// TwinCAT 3 PLC project LF_System_PLC
// ProgramVersion: 3.1.4026.22
// CompilerDefines: VISU_USEPROPERTYINFO
// libraries:
//   Tc2_MC2, * (Beckhoff Automation GmbH)
//   Tc2_Standard, * (Beckhoff Automation GmbH)
//   Tc2_System, * (Beckhoff Automation GmbH)
//   Tc3_IotBase, * (Beckhoff Automation GmbH)
//   VisuSymbols, 4.5.0.0 (System)
// project tree:
//   / GlobalTextList.TcGTLO (not stored), PlcTask.TcTTO (not stored), Visualization Manager.TcVMO (not stored)
//   GVLs/ GVL_PosKinematic.TcGVL, IFC_HW.TcGVL
//   POUs/Abfüllmodul/ FB_Abfuellmodul.TcPOU, FB_Dispenser.TcPOU (not stored), FB_EZylinder.TcPOU, FB_Vereinzelung.TcPOU (not stored)
//   POUs/ eBetriebszustand.TcDUT, FB_MqttPublisher.TcPOU, FUN_Scale.TcPOU, MAIN.TcPOU
//   POUs/Extruder/ FB_System_FlaschenFullstand.TcPOU, FB_System_Fullstand.TcPOU (not stored)
//   POUs/Förderband/ FB_System_CNV.TcPOU (not stored)
//   POUs/IoT/ FB_MQTT.TcPOU (not stored)
//   POUs/Manipulator/ FB_Manipulator.TcPOU (not stored)
//   POUs/Manipulator/Roboter/ FB_Roboter.TcPOU (not stored), FB_Roboter_Axis.TcPOU, FB_Roboter_E.TcPOU, FB_Roboter_Logik.TcPOU
//   POUs/Statusleuchte/ FB_Ampelleuchte.TcPOU, FB_Blinklicht.TcPOU
//   POUs/Transport/ FB_Foerderband.TcPOU, FB_Transport.TcPOU, FB_Transport_A.TcPOU, FB_Transport_E.TcPOU, FB_Transport_Logik.TcPOU
//   POUs/Vereinzelung/ FB_SpeicherRohr.TcPOU (not stored), FB_System_Vereinzelung.TcPOU (not stored)
//   VISUs/ Visualization.TcVIS
// real-time tasks:
//   TASK PlcTask: cycle T#10ms, priority 21, ADS port 350
//   TASK PlcTask1: cycle T#10ms, priority 22, ADS port 351
// motion (NC):
//   TASK NC-Task 1 SAF: cycle T#2ms, priority 4, ADS port 501
//   TASK NC-Task 1 SVB: cycle T#10ms, priority 8, ADS port 511
//   AXIS Band (id 1)
//     OtherSettings: AllowMotionCmdToSlave=true
//     encoder EncType=1
//     drive DrvType=5
//       Analog: TorqueSetpointScale=10, ScaleFactorActTorque=0.1
//       TimeComp: TaskDelayCycles=1
//     controller CtrType=1
//       CtrPara: PriorControlFactor=1
//         Observer: BandWidth=20
//   AXIS Extruder1 (id 2)
//     OtherSettings: AllowMotionCmdToSlave=true
//     encoder EncType=1
//     drive DrvType=5
//       Analog: TorqueSetpointScale=10, ScaleFactorActTorque=0.1
//       TimeComp: TaskDelayCycles=1
//     controller CtrType=1
//       CtrPara: PriorControlFactor=1
//         Observer: BandWidth=20
//   AXIS Extruder2 (id 3)
//     OtherSettings: AllowMotionCmdToSlave=true
//     encoder EncType=1
//     drive DrvType=5
//       Analog: TorqueSetpointScale=10, ScaleFactorActTorque=0.1
//       TimeComp: TaskDelayCycles=1
//     controller CtrType=1
//       CtrPara: PriorControlFactor=1
//         Observer: BandWidth=20
//   AXIS Extruder3 (id 4)
//     OtherSettings: AllowMotionCmdToSlave=true
//     encoder EncType=1
//     drive DrvType=5
//       Analog: TorqueSetpointScale=10, ScaleFactorActTorque=0.1
//       TimeComp: TaskDelayCycles=1
//     controller CtrType=1
//       CtrPara: PriorControlFactor=1
//         Observer: BandWidth=20
//   AXIS ManX (id 5)
//     OtherSettings: AllowMotionCmdToSlave=true
//     encoder EncType=1
//     drive DrvType=5
//       Analog: TorqueSetpointScale=10, ScaleFactorActTorque=0.1
//       TimeComp: TaskDelayCycles=1
//     controller CtrType=1
//       CtrPara: PriorControlFactor=1
//         Observer: BandWidth=20
//   AXIS ManY (id 6)
//     OtherSettings: AllowMotionCmdToSlave=true
//     encoder EncType=1
//     drive DrvType=5
//       Analog: TorqueSetpointScale=10, ScaleFactorActTorque=0.1
//       TimeComp: TaskDelayCycles=1
//     controller CtrType=1
//       CtrPara: PriorControlFactor=1
//         Observer: BandWidth=20
//   AXIS ManZ (id 7)
//     OtherSettings: AllowMotionCmdToSlave=true
//     encoder EncType=1
//     drive DrvType=5
//       Analog: TorqueSetpointScale=10, ScaleFactorActTorque=0.1
//       TimeComp: TaskDelayCycles=1
//     controller CtrType=1
//       CtrPara: PriorControlFactor=1
//         Observer: BandWidth=20
//   AXIS ManG (id 8)
//     OtherSettings: AllowMotionCmdToSlave=true
//     encoder EncType=1
//     drive DrvType=5
//       Analog: TorqueSetpointScale=10, ScaleFactorActTorque=0.1
//       TimeComp: TaskDelayCycles=1
//     controller CtrType=1
//       CtrPara: PriorControlFactor=1
//         Observer: BandWidth=20
// variable links:
//   LF_System_PLC/LF_System_PLC Instance <-> NC-Task 1 SAF/Axes/Band
//     PlcTask Inputs/IFC_HW.ax_BandMotor.NcToPlc <-> Outputs/ToPlc
//     PlcTask Outputs/IFC_HW.ax_BandMotor.PlcToNc <-> Inputs/FromPlc
//   LF_System_PLC/LF_System_PLC Instance <-> NC-Task 1 SAF/Axes/Extruder1
//     PlcTask Inputs/IFC_HW.ax_Extruder1.NcToPlc <-> Outputs/ToPlc
//     PlcTask Outputs/IFC_HW.ax_Extruder1.PlcToNc <-> Inputs/FromPlc
//   LF_System_PLC/LF_System_PLC Instance <-> NC-Task 1 SAF/Axes/Extruder2
//     PlcTask Inputs/IFC_HW.ax_Extruder2.NcToPlc <-> Outputs/ToPlc
//     PlcTask Outputs/IFC_HW.ax_Extruder2.PlcToNc <-> Inputs/FromPlc
//   LF_System_PLC/LF_System_PLC Instance <-> NC-Task 1 SAF/Axes/Extruder3
//     PlcTask Inputs/IFC_HW.ax_Extruder3.NcToPlc <-> Outputs/ToPlc
//     PlcTask Outputs/IFC_HW.ax_Extruder3.PlcToNc <-> Inputs/FromPlc
//   LF_System_PLC/LF_System_PLC Instance <-> NC-Task 1 SAF/Axes/ManG
//     PlcTask Inputs/IFC_HW.ax_ManG.NcToPlc <-> Outputs/ToPlc
//     PlcTask Outputs/IFC_HW.ax_ManG.PlcToNc <-> Inputs/FromPlc
//   LF_System_PLC/LF_System_PLC Instance <-> NC-Task 1 SAF/Axes/ManX
//     PlcTask Inputs/IFC_HW.ax_ManX.NcToPlc <-> Outputs/ToPlc
//     PlcTask Outputs/IFC_HW.ax_ManX.PlcToNc <-> Inputs/FromPlc
//   LF_System_PLC/LF_System_PLC Instance <-> NC-Task 1 SAF/Axes/ManY
//     PlcTask Inputs/IFC_HW.ax_ManY.NcToPlc <-> Outputs/ToPlc
//     PlcTask Outputs/IFC_HW.ax_ManY.PlcToNc <-> Inputs/FromPlc
//   LF_System_PLC/LF_System_PLC Instance <-> NC-Task 1 SAF/Axes/ManZ
//     PlcTask Inputs/IFC_HW.ax_ManZ.NcToPlc <-> Outputs/ToPlc
//     PlcTask Outputs/IFC_HW.ax_ManZ.PlcToNc <-> Inputs/FromPlc

// ---- POUs/eBetriebszustand.TcDUT
{attribute 'qualified_only'}
{attribute 'strict'}
{attribute 'to_string'}
TYPE eBetriebszustand :
(
	Off        := 0,   // nicht betriebsbereit
	Error      := 1,   // Fehlerbehafteter Stop
	Setup      := 2,   // Wartung
	Warning    := 3,   // nicht fehlerbehafteter, nicht geplanter Stop
	Init       := 4,   // Herstellung Betriebsbereitschaft
	Ready      := 5,   // betriebsbereit
	Production := 6,   // Betrieb
	Done       := 7,   // Betrieb abgeschlossen
	Stop       := 8
);
END_TYPE

// ---- GVLs/GVL_PosKinematic.TcGVL
{attribute 'qualified_only'}
VAR_GLOBAL
	// Home position
	pXhome : REAL := 29;
	pYhome : REAL := 145.5;
	pZhome : REAL := 45;
	
	// Conveyor position
	pXconv : REAL := 29;
	pYconv : REAL := 145.5;
	pZconv : REAL := 130;
	
	//Scale position
	pXscale : REAL := 36;
	pYscale : REAL := 7.5;
	pZscale : REAL := 131.5;
	
	// Heating position
	pXheat : REAL := 218.5;
	pYheat : REAL := 7;
	pZheat : REAL := 159;
	
	// Storage position
	pX1stor : REAL := 107;
	pX2stor : REAL := 158.7;
	pX3stor : REAL := 209.3;
	pX4stor : REAL := 260.3;
	pYstor : REAL := 139;
	pZstor : REAL := 120;
	
	// Z offset height
	pZoff : REAL := 45;
END_VAR

// ---- GVLs/IFC_HW.TcGVL
// In dieser GVL werden alle Variablen deklariert die auf die realen Klemmen zugreifen
VAR_GLOBAL
	
	// Allgemeine Variablen fur MAIN und HMI
		bEnable		AT%I*	: BOOL;			// Enable Factory (HMI Production Umgebung)
		bExecute	AT%I*	: BOOL;			// Startsignal	(Start Knopf Konsole)
		bStop				: BOOL;			// Stop Variable (interne Variable um FB's zu stoppen)
		
	// Station Statusampel	
		bAmpelRot 	AT%Q* 	: BOOL;			// Signal-LED Rot
		bAmpelGelb 	AT%Q* 	: BOOL;			// Signal-LED Gelb
		bAmpelGrun 	AT%Q* 	: BOOL;			// Signal-LED Grun
			
	// Station Vereinzelung
		bEinzelSens1 	AT%I*	: BOOL;					// Separation Sensor 1 (Kammer)
		bEinzelSens2 	AT%I*	: BOOL;					// Separation Sensor 2 (Rohr)
		bEinzelSens3 	AT%I*	: BOOL;					// Separation Sensor 3 (Flasche auf Kopf)
		bR1AKT1 		AT%Q* 	: BOOL := FALSE;		// Relais 1 Aktor 1 (Schleuse Oben öffnen)
		bR2AKT1 		AT%Q* 	: BOOL := TRUE; 		// Relais 2 Aktor 1 (Schleuse Oben schließen)
		bR1AKT2 		AT%Q* 	: BOOL := FALSE;		// Relais 1 Aktor 2 (Schleuse Unten öffne)
		bR2AKT2 		AT%Q* 	: BOOL := TRUE;			// Relais 2 Aktor 2	(Schleuse Unten schließen)
	
	// Station Forderband
		bBandSens1 	AT %I*	: BOOL;		// Forderband Sensor 1 (Extruder 1)
		bBandSens2	AT %I*	: BOOL;		// Forderband Sensor 2 (Extruder 2)
		bBandSens3 	AT %I*	: BOOL;		// Forderband Sensor 3 (Extruder 3)
		bBandSens4 	AT %I*	: BOOL;		// Forderband Sensor 4 (Übergabe Roboter)
		bBandHub1 	AT %Q*	: BOOL;		// Forderband Hubmagnet 1 (Schleuse Extruder 1)
		bBandHub2 	AT %Q*	: BOOL;		// Forderband Hubmagnet 1 (Schleuse Extruder 2)
		bBandHub3 	AT %Q*	: BOOL;		// Forderband Hubmagnet 1 (Schleuse Extruder 3)
		
		ax_Extruder1 	: AXIS_REF;		// Forderband NC-Achse Extruder 1
		ax_Extruder2 	: AXIS_REF;		// Forderband NC-Achse Extruder 2
		ax_Extruder3 	: AXIS_REF;		// Forderband NC-Achse Extruder 3
		ax_BandMotor 	: AXIS_REF;		// Forderband NC-Achse Band
		
		iBandFullmenge1		: INT := 1;	// in Gramm (Soll Füllmenge Extruder 1)
		iBandFullmenge2		: INT := 1;	// in Gramm (Soll Füllmenge Extruder 2)
		iBandFullmenge3		: INT := 1;	// in Gramm (Soll Füllmenge Extruder 3)
		
	//Füllstandsüberwachung
		iFillSens1 AT%I*	: UINT;		// Füllstandssensor im Granulatspeicher 1
		iFillSens2 AT%I*	: UINT;		// Füllstandssensor im Granulatspeicher 2
		iFillSens3 AT%I*	: UINT;		// Füllstandssensor im Granulatspeicher 3
		
		rFillLevelPercent1	: REAL;		// Füllstand im Granulatspeicher 1 in %
		rFillLevelGramm1	: REAL;		// Füllstand im Granulatspeicher 1 in g
		rFillLevelPercent2	: REAL;		// Füllstand im Granulatspeicher 2 in %
		rFillLevelGramm2	: REAL;		// Füllstand im Granulatspeicher 2 in g
		rFillLevelPercent3	: REAL;		// Füllstand im Granulatspeicher 3 in %
		rFillLevelGramm3	: REAL;		// Füllstand im Granulatspeicher 3 in g
		
		rMaxFillLevel 		: REAL := 375;	// Kalibrierter Füllstand für 10% * 10
		
	// Station Waage
		sWaageNachricht		: STRING;	// Nachricht von Wagezelle (fur virtuelle Inbetriebnahme notig)
		bWaageNull			: BOOL;		// TARA Waage (Waage auf Null setzen)
		iWaageMesswert		: INT;		// Messwert der Waage
		
	// Station Behalteridentifikation
		bIdSensorTrager		: BOOL;		// Sensor bei Erkennung eines Datentrager
		sIdNachricht		: STRING;	// Nachricht von RFID-System (fur virtuelle Inbetriebnahme notig)
		sSeriennummer		: STRING;	// Seriennummer RFID-Tag
		
	//Temperierstation
		bVentilator1 	AT %Q*	: BOOL;		// Ventilator 1
		bVentilator2 	AT %Q*	: BOOL;		// Ventilator 2
		bVentilator3 	AT %Q*	: BOOL;		// Ventilator 3
		
		iTempSens1 		AT%I*	: UINT;		// Temperatursensor 1
		iTempSens2 		AT%I*	: UINT;		// Temperatursensor 2
		iHeizpatrone 	AT%Q*	: UINT;		// Heizpatronen
		
		iMaxTemp				: UINT := 5500;		// in °C * 100
		
	// Station Manipulator
		bManEndXmin 		AT%I* 	: BOOL := TRUE;		// Manipulator min Endschalter Achse x
		bManEndYmin 		AT%I* 	: BOOL := TRUE;		// Manipulator min Endschalter Achse y
		bManEndZmin 		AT%I* 	: BOOL := TRUE;		// Manipulator min Endschalter Achse z
		bManEndGmin 		AT%I* 	: BOOL := TRUE;		// Manipulator min Endschalter Achse Gripper
		bManEndXmax 		AT%I* 	: BOOL := TRUE;		// Manipulator max Endschalter Achse x
		bManEndYmax 		AT%I* 	: BOOL := TRUE;		// Manipulator max Endschalter Achse y
		bManEndZmax 		AT%I* 	: BOOL := TRUE;		// Manipulator max Endschalter Achse z
		bManEndGmax 		AT%I* 	: BOOL := TRUE;		// Manipulator max Endschalter Achse Gripper
		bManBrakeZ			AT%Q*	: BOOL := FALSE;	// Bremse Achse z
		
		ax_ManX			: AXIS_REF;			// Manipulator NC-Achse x
		ax_ManY			: AXIS_REF;			// Manipulator NC-Achse y
		ax_ManZ			: AXIS_REF;			// Manipulator NC-Achse z
		ax_ManG			: AXIS_REF; 		// Manipulator NC-Achse Gripper
		
		bGripperClosed		AT%Q*	: BOOL; 			// signal if gripper is closed ONLY USED IN SIM
			// --- Für die Unity-Simulation (TeachingFactory) benötigt ---
	BandExtruder1_Enable AT%Q* : BOOL;
	BandExtruder1_Velocity AT%Q* : LREAL;
	BandExtruder2_Enable AT%Q* : BOOL;
	BandExtruder2_Velocity AT%Q* : LREAL;
	BandExtruder3_Enable AT%Q* : BOOL;
	BandExtruder3_Velocity AT%Q* : LREAL;
	BandMotor_Enable AT%Q* : BOOL;
	BandMotor_Velocity AT%Q* : LREAL;

	EinzelActor1_1 AT%Q* : BOOL;
	EinzelActor1_2 AT%Q* : BOOL;
	EinzelActor2_1 AT%Q* : BOOL;
	EinzelActor2_2 AT%Q* : BOOL;

	ManAchseX_Enable AT%Q* : BOOL;
	ManAchseX_Homed AT%I* : BOOL;
	ManAchseX_Position AT%Q* : LREAL;
	ManAchseX_Velocity AT%Q* : LREAL;
	ManAchseY_Enable AT%Q* : BOOL;
	ManAchseY_Homed AT%I* : BOOL;
	ManAchseY_Position AT%Q* : LREAL;
	ManAchseY_Velocity AT%Q* : LREAL;
	ManAchseZ_Enable AT%Q* : BOOL;
	ManAchseZ_Homed AT%I* : BOOL;
	ManAchseZ_Position AT%Q* : LREAL;
	ManAchseZ_Velocity AT%Q* : LREAL;
	ManAchseGrip_Enable AT%Q* : BOOL;
	ManAchseGrip_Homed AT%I* : BOOL;
	ManAchseGrip_Position AT%Q* : LREAL;
	ManAchseGrip_Velocity AT%Q* : LREAL;

	bGripperClosed_doNotUse AT%Q* : BOOL;

END_VAR

// ---- POUs/MAIN.TcPOU
PROGRAM MAIN
VAR
	fb_Ampelleuchte :FB_Ampelleuchte;	
	fb_Abfuellmodul :FB_Abfuellmodul;
	fb_Manipulator :FB_Manipulator;

	nState :INT :=0;

	fb_MQTT :FB_MQTT;

	fb_MqttPublisher : FB_MqttPublisher;
	FB_System_FlaschenFullstand : FB_System_Flaschenfullstand;
END_VAR

	
fb_Ampelleuchte(eState:= , bAmpelGruen_out=> IFC_HW.bAmpelGrun, bAmpelRot_out=> IFC_HW.bAmpelRot, bAmpelGelb_out=> IFC_HW.bAmpelGelb);

fb_Abfuellmodul(bEnable:= , bExecute:= , eState=> ); 
fb_Manipulator(bEnable:= , bExecute:= , bGripperClosed=> IFC_HW.bGripperClosed, eState=> );

IF fb_Abfuellmodul.eState = eBetriebszustand.Init OR fb_Manipulator.eState = eBetriebszustand.Init THEN
	fb_Ampelleuchte.eState := eBetriebszustand.init;
ELSIF fb_Abfuellmodul.eState = eBetriebszustand.ready AND fb_Manipulator.eState = eBetriebszustand.ready THEN
	fb_Ampelleuchte.eState := eBetriebszustand.ready;
ELSIF fb_Abfuellmodul.eState = eBetriebszustand.production OR fb_Manipulator.eState = eBetriebszustand.Production THEN
	fb_Ampelleuchte.eState := eBetriebszustand.Production;
ELSIF fb_Abfuellmodul.eState = eBetriebszustand.off AND fb_Manipulator.eState = eBetriebszustand.off THEN
	fb_Ampelleuchte.eState := eBetriebszustand.off;
ELSE 
	fb_Ampelleuchte.eState := eBetriebszustand.Warning;
END_IF



IF NOT IFC_HW.bEnable THEN
	nState :=0;
END_IF
CASE nState Of
	0://off
	fb_Abfuellmodul.bEnable :=FALSE;
	fb_Manipulator.bEnable :=FALSE;
	
	IF IFC_HW.bEnable THEN
		nstate:=1;
	END_IF
	
	1: //init
	fb_Abfuellmodul.bEnable :=TRUE;
	fb_Manipulator.bEnable :=TRUE;
	
	IF fb_Abfuellmodul.eState = eBetriebszustand.Ready AND fb_Manipulator.eState = eBetriebszustand.Ready THEN
		nState:=2;
	END_IF
	
	2: //ready
	IF IFC_HW.bExecute AND iFC_HW.bEinzelSens1 THEN
		nstate :=21;
	END_IF
	IF NOT iFC_HW.bEinzelSens2 AND NOT iFC_HW.bEinzelSens1 THEN
		fb_Abfuellmodul.bEnable :=FALSE;
		nState :=1;
	END_IF
	
	21: //bottle
	fb_Abfuellmodul.bExecute :=TRUE;
	
	IF fb_Abfuellmodul.eState = eBetriebszustand.Done THEN
		fb_Abfuellmodul.bExecute :=FALSE;
		nstate :=22;
	END_IF
	
	22: //mani
	fb_Manipulator.bExecute :=TRUE;
	
	IF fb_Manipulator.eState = eBetriebszustand.Done THEN
		fb_Manipulator.bExecute :=FALSE;
		nState :=23;
	END_IF
	
	23://done
	IF NOT IFC_HW.bExecute THEN
		nState:=2;
	END_IF
END_CASE
FB_System_FlaschenFullstand(
    rFilling1 := IFC_HW.ax_Extruder1.NcToPlc.ActPos,
    rFilling2 := IFC_HW.ax_Extruder2.NcToPlc.ActPos,
    rFilling3 := IFC_HW.ax_Extruder3.NcToPlc.ActPos,
    Reset := ,
    rPcntFillLevelOut => ,
    iFillLevel1Out => ,
    iFillLevel2Out => ,
    iFillLevel3Out =>
);

fb_MqttPublisher(
    bEnableMqtt := IFC_HW.bEnable,

    iBandFullmenge1 := IFC_HW.iBandFullmenge1,

    bEnable := IFC_HW.bEnable,
    bExecute := IFC_HW.bExecute,

    bEinzelSens1 := IFC_HW.bEinzelSens1,
    bEinzelSens2 := IFC_HW.bEinzelSens2,
    bEinzelSens3 := IFC_HW.bEinzelSens3,

    bBandSens1 := IFC_HW.bBandSens1,
    bBandSens2 := IFC_HW.bBandSens2,
    bBandSens3 := IFC_HW.bBandSens3,
    bBandSens4 := IFC_HW.bBandSens4,

    rPcntFillLevel := fb_System_FlaschenFullstand.rPcntFillLevelOut,
    iFillLevel1 := fb_System_FlaschenFullstand.iFillLevel1Out,
    iFillLevel2 := fb_System_FlaschenFullstand.iFillLevel2Out,
    iFillLevel3 := fb_System_FlaschenFullstand.iFillLevel3Out,

    bConnected => ,
    bError => ,
    hrErrorCode =>
);

fb_MqttPublisher(
    bEnableMqtt := IFC_HW.bEnable,

    iBandFullmenge1 := IFC_HW.iBandFullmenge1,

    bEnable := IFC_HW.bEnable,
    bExecute := IFC_HW.bExecute,

    bEinzelSens1 := IFC_HW.bEinzelSens1,
    bEinzelSens2 := IFC_HW.bEinzelSens2,
    bEinzelSens3 := IFC_HW.bEinzelSens3,

    bBandSens1 := IFC_HW.bBandSens1,
    bBandSens2 := IFC_HW.bBandSens2,
    bBandSens3 := IFC_HW.bBandSens3,
    bBandSens4 := IFC_HW.bBandSens4,

    rPcntFillLevel := fb_System_FlaschenFullstand.rPcntFillLevelOut,
    iFillLevel1 := fb_System_FlaschenFullstand.iFillLevel1Out,
    iFillLevel2 := fb_System_FlaschenFullstand.iFillLevel2Out,
    iFillLevel3 := fb_System_FlaschenFullstand.iFillLevel3Out,

    bConnected => ,
    bError => ,
    hrErrorCode =>
);

END_PROGRAM

// ---- POUs/Statusleuchte/FB_Ampelleuchte.TcPOU
FUNCTION_BLOCK FB_Ampelleuchte
VAR_INPUT
	eState : eBetriebszustand;
END_VAR
VAR_OUTPUT

	
	bAmpelGruen_out :BOOL;
	bAmpelRot_out :BOOL;
	bAmpelGelb_out :BOOL;
	
END_VAR
VAR
	fb_BlinklichtGr :FB_Blinklicht;
	fb_BlinklichtRt :FB_Blinklicht;
	fb_BlinklichtGb :FB_Blinklicht;
	AmpelGruenblinken:BOOL;
	AmpelRotblinken :BOOL;
	AmpelGelbblinken :BOOL;
	bAmpelGruen :BOOL;
	bAmpelRot :BOOL;
	bAmpelGelb :BOOL;
END_VAR

CASE eState OF
	0: //OFF nicht Betriebsbereit
	//keine Lampe leuchtet
	bAmpelGruen :=FALSE;
	bAmpelRot :=FALSE;
	bAmpelGelb :=FALSE;
	AmpelGruenblinken:=FALSE;
	AmpelRotblinken :=FALSE;
	AmpelGelbblinken :=FALSE;
	
	1: //Error Fehlerbehafteter Stop (Sicherheitssteuerung)
	//Rote Lampe Leuchtet 
	bAmpelGruen :=FALSE;
	bAmpelRot :=TRUE;
	bAmpelGelb :=FALSE;
	AmpelGruenblinken:=FALSE;
	AmpelRotblinken :=FALSE;
	AmpelGelbblinken :=FALSE;
	
	2: //Setup Wartung
	//Rot und Gelb blinkt
	bAmpelGruen :=FALSE;
	bAmpelRot :=FALSE;
	bAmpelGelb :=FALSE;
	AmpelGruenblinken:=FALSE;
	AmpelRotblinken :=TRUE;
	AmpelGelbblinken :=TRUE;
	
	3: //Warning Nicht Fehlerbehafteter nicht geplanter Stop
	//Gelb blinken
	bAmpelGruen :=FALSE;
	bAmpelRot :=FALSE;
	bAmpelGelb :=FALSE;
	AmpelGruenblinken:=FALSE;
	AmpelRotblinken :=FALSE;
	AmpelGelbblinken :=TRUE;
	
	4: //Init Herstellung Betriebsbereitschaft
	//Gelb Grün blinkt
	bAmpelGruen :=FALSE;
	bAmpelRot :=FALSE;
	bAmpelGelb :=FALSE;
	AmpelGruenblinken:=TRUE;
	AmpelRotblinken :=FALSE;
	AmpelGelbblinken :=TRUE;
	
	5: //Ready Betriebsbereit
	//Grün blinkt
	bAmpelGruen :=FALSE;
	bAmpelRot :=FALSE;
	bAmpelGelb :=FALSE;
	AmpelGruenblinken:=TRUE;
	AmpelRotblinken :=FALSE;
	AmpelGelbblinken :=FALSE;
	
	6: //Production Betrieb
	//Grün leuchtet
	bAmpelGruen :=TRUE;
	bAmpelRot :=FALSE;
	bAmpelGelb :=FALSE;
	AmpelGruenblinken:=FALSE;
	AmpelRotblinken :=FALSE;
	AmpelGelbblinken :=FALSE;
	
	7: //Done Betrieb abgeschlossen 
	//Grün Gelb leuchten
	bAmpelGruen :=TRUE;
	bAmpelRot :=FALSE;
	bAmpelGelb :=TRUE;
	AmpelGruenblinken:=FALSE;
	AmpelRotblinken :=FALSE;
	AmpelGelbblinken :=FALSE;
	
	8: //Stop
	//Rot blinken
	bAmpelGruen :=FALSE;
	bAmpelRot :=FALSE;
	bAmpelGelb :=FALSE;
	AmpelGruenblinken:=FALSE;
	AmpelRotblinken :=TRUE;
	AmpelGelbblinken :=FALSE;
END_CASE

fb_BlinklichtGb(bStartStop:= AmpelGelbblinken, tPeriod:= T#1S , bBlink=> );
fb_BlinklichtGr(bStartStop:= AmpelGruenblinken, tPeriod:= T#1S, bBlink=> );
fb_BlinklichtRt(bStartStop:= AmpelRotblinken, tPeriod:= T#1S, bBlink=> );

IF fb_BlinklichtGb.bBlink OR bAmpelGelb THEN
	bAmpelGelb_out :=TRUE;
ELSE
	bAmpelGelb_out :=FALSE;
END_IF
IF fb_BlinklichtGr.bBlink OR bAmpelGruen THEN
	bAmpelGruen_out :=TRUE;
ELSE
	bAmpelGruen_out :=FALSE;
END_IF
IF fb_BlinklichtRt.bBlink OR bAmpelRot THEN
	bAmpelRot_out :=TRUE;
ELSE
	bAmpelRot_out :=FALSE;
END_IF

END_FUNCTION_BLOCK

// ---- POUs/Statusleuchte/FB_Blinklicht.TcPOU
FUNCTION_BLOCK FB_Blinklicht
VAR_INPUT
	bStartStop :BOOL;
	tPeriod :TIME := T#1s;
	
END_VAR
VAR_OUTPUT
	bBlink :BOOL;
	
END_VAR
VAR
	fbTON :TON;
	fbRtrig :R_Trig;
	bEinAus :BOOL := 0;
END_VAR

fbRtrig(CLK:= bStartStop, Q=> );

IF fbRtrig.Q THEN
	bEinAus:= NOT bEinAus;
END_IF


//fbTON.IN := bBlink AND NOT fbTON.Q;
//fbTON.PT:=T#1S;

fbTON(in:=bEinAus AND NOT fbTON.Q , PT:= tPeriod, Q=>,ET=>);

IF fbTON.ET<=fbTON.PT/2 THEN
	bBlink := FALSE;
ELSIF fbTON.ET>fbTON.PT/2 THEN
	bBlink := TRUE;
END_IF

(*IF NOT bBlink THEN
	bLEDrot := FALSE;
END_IF
*)

IF NOT bStartStop THEN
	bBlink :=FALSE;
END_IF

END_FUNCTION_BLOCK

// ---- POUs/Abfüllmodul/FB_Abfuellmodul.TcPOU
FUNCTION_BLOCK FB_Abfuellmodul
VAR_INPUT
	bEnable :BOOL;
	bExecute :BOOL;
END_VAR
VAR_OUTPUT
	eState :eBetriebszustand;
END_VAR
VAR
	fb_Vereinzelung :FB_Vereinzelung;
	fb_Transport : FB_Transport;
	fb_Dispenser1 :FB_Dispenser;
	fb_Dispenser2 :FB_Dispenser;
	fb_Dispenser3 :FB_Dispenser;
	fb_EZylinder1 : FB_EZylinder;
	fb_EZylinder2 : FB_EZylinder;

	
	nState :INT;
	nStation :INT;
END_VAR

fb_Vereinzelung(
	bEnable:= , 
	bExecute:= , 
	bSens1:= IFC_HW.bEinzelSens1, 
	bSens2:= IFC_HW.bEinzelSens2, 
	bSens3:= IFC_HW.bEinzelSens3, 
	bSens4:= IFC_HW.bBandSens1, 
	eState=> , 
	bGate1=> fb_EZylinder1.bGate, 
	bGate2=> fb_EZylinder2.bGate);
	
fb_Transport(
	bEnable:= , 
	bExecute:= , 
	nStation:= nStation, 
	bSens1:= IFC_HW.bBandSens1, 
	bSens2:= IFC_HW.bBandSens2, 
	bSens3:= IFC_HW.bBandSens3, 
	bSens4:= IFC_HW.bBandSens4, 
	eState=> , 
	bStopper1=> IFC_HW.bBandHub1, 
	bStopper2=> IFC_HW.bBandHub2, 
	bStopper3=> IFC_HW.bBandHub3, 
	ax:= IFC_HW.ax_BandMotor);
	
fb_Dispenser1(
	bEnable:= , 
	bExecute:= , 
	rDistance:= IFC_HW.iBandFullmenge1*20, 
	eState=> , 
	ax:= IFC_HW.ax_Extruder1);
fb_Dispenser2(
	bEnable:= , 
	bExecute:= , 
	rDistance:= IFC_HW.iBandFullmenge1*20, 
	eState=> , 
	ax:= IFC_HW.ax_Extruder2);
fb_Dispenser3(
	bEnable:= , 
	bExecute:= , 
	rDistance:= IFC_HW.iBandFullmenge1*20, 
	eState=> , 
	ax:= IFC_HW.ax_Extruder3);
	
fb_EZylinder1(bGate:= , bError:= , bR1=> IFC_HW.bR1AKT1, bR2=> IFC_HW.bR2AKT1);
fb_EZylinder2(bGate:= , bError:= , bR1=> IFC_HW.bR1AKT2, bR2=> IFC_HW.bR2AKT2);


IF NOT bEnable THEN 
	nState :=0;
END_IF


CASE nState OF
	0: // Off
	eState := eBetriebszustand.Off;
	
	fb_Vereinzelung.bEnable:=FALSE;
	fb_Transport.bEnable :=FALSE;
	fb_Dispenser1.bEnable :=FALSE;
	fb_Dispenser2.bEnable :=FALSE;
	fb_Dispenser3.bEnable :=FALSE;
	fb_Vereinzelung.bExecute :=FALSE;
	fb_Transport.bExecute :=FALSE;
	fb_Dispenser1.bExecute :=FALSE;
	fb_Dispenser2.bExecute :=FALSE;
	fb_Dispenser3.bExecute :=FALSE;
	
	IF bEnable THEN
		nstate :=10;
	END_IF
	
	10:// Init
	eState := eBetriebszustand.Init;
	
	fb_Vereinzelung.bEnable:=TRUE;
	fb_Transport.bEnable :=TRUE;
	fb_Dispenser1.bEnable :=TRUE;
	fb_Dispenser2.bEnable :=TRUE;
	fb_Dispenser3.bEnable :=TRUE;
	fb_Vereinzelung.bExecute :=FALSE;
	fb_Transport.bExecute :=FALSE;
	fb_Dispenser1.bExecute :=FALSE;
	fb_Dispenser2.bExecute :=FALSE;
	fb_Dispenser3.bExecute :=FALSE;
	
	IF (fb_Vereinzelung.eState = eBetriebszustand.Ready) AND (fb_Transport.eState = eBetriebszustand.Ready) AND (fb_Dispenser1.eState = eBetriebszustand.Ready) AND (fb_Dispenser2.eState = eBetriebszustand.Ready) AND (fb_Dispenser3.eState = eBetriebszustand.Ready)THEN
		nstate :=20;
	END_IF
	
	20:// Ready
	eState := eBetriebszustand.Ready;
	
	fb_Vereinzelung.bEnable:=TRUE;
	fb_Transport.bEnable :=TRUE;
	fb_Dispenser1.bEnable :=TRUE;
	fb_Dispenser2.bEnable :=TRUE;
	fb_Dispenser3.bEnable :=TRUE;
	fb_Vereinzelung.bExecute :=FALSE;
	fb_Transport.bExecute :=FALSE;
	fb_Dispenser1.bExecute :=FALSE;
	fb_Dispenser2.bExecute :=FALSE;
	fb_Dispenser3.bExecute :=FALSE;
	
	IF bExecute THEN
		nState:=30;
	END_IF
	
	30:// Start
	eState := eBetriebszustand.Production;
	
	fb_Vereinzelung.bExecute :=TRUE;
	fb_Transport.bExecute :=TRUE;
	fb_Dispenser1.bExecute :=FALSE;
	fb_Dispenser2.bExecute :=FALSE;
	fb_Dispenser3.bExecute :=FALSE;
	nStation :=1;
	
	IF (fb_Vereinzelung.eState = eBetriebszustand.Done) AND (fb_Transport.eState = eBetriebszustand.Done) THEN
		nstate :=31;
	END_IF
	
	31:// Dispenser1
	eState := eBetriebszustand.Production;
	
	fb_Vereinzelung.bExecute :=FALSE;
	fb_Transport.bExecute :=FALSE;
	fb_Dispenser1.bExecute :=TRUE;
	fb_Dispenser2.bExecute :=FALSE;
	fb_Dispenser3.bExecute :=FALSE;
	nStation :=1;
	
	IF fb_Dispenser1.eState = eBetriebszustand.Done THEN
		nState :=32;
	END_IF
	
	32:// Bewegung zu Dispenser2
	eState := eBetriebszustand.Production;
	
	nStation :=2;
	fb_Vereinzelung.bExecute :=FALSE;
	fb_Transport.bExecute :=TRUE;
	fb_Dispenser1.bExecute :=FALSE;
	fb_Dispenser2.bExecute :=FALSE;
	fb_Dispenser3.bExecute :=FALSE;
	
	IF fb_Transport.eState = eBetriebszustand.Done THEN
		nState :=33;
	END_IF
	
	33:// Dispenser2
	eState := eBetriebszustand.Production;
	
	fb_Vereinzelung.bExecute :=FALSE;
	fb_Transport.bExecute :=FALSE;
	fb_Dispenser1.bExecute :=FALSE;
	fb_Dispenser2.bExecute :=TRUE;
	fb_Dispenser3.bExecute :=FALSE;
	nStation :=2;
	
	IF fb_Dispenser2.eState = eBetriebszustand.Done THEN
		nState :=34;
	END_IF
		
	34:// Bewegung zu Dispenser3
	eState := eBetriebszustand.Production;
	
	nStation :=3;
	fb_Vereinzelung.bExecute :=FALSE;
	fb_Transport.bExecute :=TRUE;
	fb_Dispenser1.bExecute :=FALSE;
	fb_Dispenser2.bExecute :=FALSE;
	fb_Dispenser3.bExecute :=FALSE;
	
	IF fb_Transport.eState = eBetriebszustand.Done THEN
		nState :=35;
	END_IF
	
	35:// Dispenser3
	eState := eBetriebszustand.Production;
	
	fb_Vereinzelung.bExecute :=FALSE;
	fb_Transport.bExecute :=FALSE;
	fb_Dispenser1.bExecute :=FALSE;
	fb_Dispenser2.bExecute :=FALSE;
	fb_Dispenser3.bExecute :=TRUE;
	nStation :=3;
	
	IF fb_Dispenser3.eState = eBetriebszustand.Done THEN
		nState :=36;
	END_IF
	
	36:// Abholstation
	eState := eBetriebszustand.Production;
	
	nStation :=4;
	fb_Vereinzelung.bExecute :=FALSE;
	fb_Transport.bExecute :=TRUE;
	fb_Dispenser1.bExecute :=FALSE;
	fb_Dispenser2.bExecute :=FALSE;
	fb_Dispenser3.bExecute :=FALSE;
		
	IF fb_Transport.eState = eBetriebszustand.Done THEN
		nState :=40;
	END_IF 
	
	40:// Done
	eState := eBetriebszustand.Done;
	
	fb_Vereinzelung.bExecute :=FALSE;
	fb_Transport.bExecute :=FALSE;
	fb_Dispenser1.bExecute :=FALSE;
	fb_Dispenser2.bExecute :=FALSE;
	fb_Dispenser3.bExecute :=FALSE;
	
	IF not bExecute THEN
		nState :=20;
	END_IF
	
	
END_CASE

END_FUNCTION_BLOCK

// ---- POUs/Transport/FB_Transport.TcPOU
FUNCTION_BLOCK FB_Transport
VAR_INPUT
	bEnable :BOOL;
	bExecute :BOOL;
	nStation :INT := 1;
	//Hardweare Eingänge
	bSens1 :BOOL;
	bSens2 :BOOL;
	bSens3 :BOOL;
	bSens4 :BOOL;
END_VAR
VAR_OUTPUT
	eState :eBetriebszustand;
	bStopper1 :BOOL;
	bStopper2 :BOOL;
	bStopper3 :BOOL;
END_VAR
VAR
	fb_TransportE :FB_Transport_E;
	fb_TransportLogik :FB_Transport_Logik;
	fb_TransportBand :FB_Foerderband;
	fb_TransportA :FB_Transport_A;
END_VAR
VAR_IN_OUT
	//Achsen Ref
	ax : AXIS_REF;
END_VAR

//nur Eingänge werden beschreiben
fb_TransportE(
	bSens1:= bSens1, 
	bSens2:= bSens2, 
	bSens3:= bSens3, 
	bSens4:= bSens4, 
	bStation1=> , 
	bStation2=> , 
	bStation3=> , 
	bStation4=> );
	
fb_TransportLogik(
	bEnable:= bEnable, 
	bExecute:= bExecute, 
	eStateE:= fb_TransportBand.eState, 
	nStation:= nStation, 
	bStation1:= fb_TransportE.bStation1, 
	bStation2:= fb_TransportE.bStation2, 
	bStation3:= fb_TransportE.bStation3, 
	bStation4:= fb_TransportE.bStation4,
	bEnableA=> , 
	bExecuteA=> , 
	bStopA=> , 
	eStateA=> eState, 
	bStop1=> , 
	bStop2=> , 
	bStop3=> );
	
	
fb_TransportBand(
	bEnable:= fb_TransportLogik.bEnableA, 
	bExecute:= fb_TransportLogik.bExecuteA, 
	bHalt:= fb_TransportLogik.bStopA, 
	eState=> , 
	ax:= ax);
	
	
fb_TransportA(
	bStop1:= fb_TransportLogik.bStop1, 
	bStop2:= fb_TransportLogik.bStop2, 
	bStop3:= fb_TransportLogik.bStop3, 
	bStopper1=> bStopper1, 
	bStopper2=> bStopper2, 
	bStopper3=> bStopper3);

END_FUNCTION_BLOCK

// ---- POUs/Transport/FB_Transport_E.TcPOU
FUNCTION_BLOCK FB_Transport_E
VAR_INPUT
	//Hardware Singale
	bSens1 :BOOL;
	bSens2 :BOOL;
	bSens3 :BOOL;
	bSens4 :BOOL;
END_VAR
VAR_OUTPUT
	bStation1 :BOOL;
	bStation2 :BOOL;
	bStation3 :BOOL;
	bStation4 :BOOL;
END_VAR
VAR
END_VAR

bStation1 :=bSens1;
bStation2 :=bSens2;
bStation3 :=bSens3;
bStation4 :=bSens4;

END_FUNCTION_BLOCK

// ---- POUs/Transport/FB_Transport_Logik.TcPOU
FUNCTION_BLOCK FB_Transport_Logik
VAR_INPUT
	bEnable :BOOL;
	bExecute :BOOL;
	eStateE :eBetriebszustand;
	nStation :INT;
	//Logik -> Hardware Signale
	bStation1 :BOOL;
	bStation2 :BOOL;
	bStation3 :BOOL;
	bStation4 :BOOL;
END_VAR
VAR_OUTPUT
	bEnableA :BOOL;
	bExecuteA :BOOL;
	bStopA :BOOL;
	eStateA :eBetriebszustand;
	
	//Hardware Singale ->Logik
	bStop1 :BOOL;
	bStop2 :BOOL;
	bStop3 :BOOL;
END_VAR
VAR
	nState :INT;
	
END_VAR


IF NOT bEnable THEN
	nState :=0;
END_IF

CASE nState OF 
	0: //off
	eStateA:= eBetriebszustand.Off;
	bEnableA :=FALSE;
	bExecuteA :=FALSE;
	bStopA :=FALSE;
	bStop1 :=FALSE;
	bStop2 :=FALSE;
	bStop3 :=FALSE;
	
	IF bEnable THEN 
		nState :=1;
	END_IF

	1: //init
	eStateA:=eBetriebszustand.Init;
	bEnableA :=TRUE;
	bExecuteA :=FALSE;
	bStopA :=FALSE;
	bStop1 :=FALSE;
	bStop2 :=FALSE;
	bStop3 :=FALSE;
	
	IF eStateE = eBetriebszustand.Ready THEN
		nState :=2;
	END_IF
	
	2: //Ready
	eStateA:=eBetriebszustand.Ready;
	bEnableA :=TRUE;
	bExecuteA :=FALSE;
	bStopA :=FALSE;
	bStop1 :=FALSE;
	bStop2 :=FALSE;
	bStop3 :=FALSE;
	
	IF bExecute THEN
		nState :=3;
	END_IF
	
	3: //Förderband Start
	eStateA:=eBetriebszustand.Production;
	bExecuteA :=TRUE;
	
	IF (nStation-1) = 1 THEN
		bStop1 :=TRUE;
	ELSIF (nStation-1) = 2 THEN
		bStop2 :=TRUE;		
	ELSIF (nStation-1) = 3 THEN
		bStop3 :=TRUE;		
	END_IF
	
	IF (bStation1 AND (nStation =1)) OR (bStation2 AND (nStation =2)) OR (bStation3 AND (nStation =3)) OR (bStation4 AND (nStation =4))THEN
		nState :=4;
	END_IF
	
	4: //Förderband stop
	eStateA:=eBetriebszustand.Production;
	bExecuteA := FALSE;
	bStopA := TRUE;
	bStop1 :=FALSE;
	bStop2 :=FALSE;
	bStop3 :=FALSE;
	
	IF eStateE = eBetriebszustand.Done THEN
		nState :=5;
	END_IF
	
	5: //Done
	eStateA:=eBetriebszustand.Done;
	
	IF NOT bExecute THEN
		nState :=2;
	END_IF
END_CASE

END_FUNCTION_BLOCK

// ---- POUs/Transport/FB_Foerderband.TcPOU
FUNCTION_BLOCK FB_Foerderband
VAR_INPUT
	bEnable :BOOL;
	bExecute :BOOL;
	bHalt :BOOL;
END_VAR
VAR_OUTPUT
	eState :eBetriebszustand;
END_VAR
VAR
	nState:INT :=0;
	mc_Reset :MC_Reset;
	mc_Velocity :MC_MoveVelocity;
	mc_Halt :MC_Halt;
	mc_Power :MC_Power;
	Timer :TON;
END_VAR
VAR_IN_OUT
	ax : Axis_Ref;
END_VAR

ax.ReadStatus();
mc_Reset(
	Axis:= ax, 
	Execute:= , 
	Done=> , 
	Busy=> , 
	Error=> , 
	ErrorID=> );
	
mc_Power(
	Axis:= ax, 
	Enable:= , 
	Enable_Positive:= , 
	Enable_Negative:= , 
	Override:= , 
	BufferMode:= , 
	Options:= , 
	Status=> , 
	Busy=> , 
	Error=> , 
	ErrorID=> );
	
mc_Velocity(
	Axis:= ax, 
	Execute:= , 
	Velocity:= 30, 
	Acceleration:= 60, 
	Deceleration:= 60, 
	Jerk:= , 
	Direction:= MC_Positive_Direction, 
	BufferMode:= , 
	Options:= , 
	InVelocity=> , 
	Busy=> , 
	Active=> , 
	CommandAborted=> , 
	Error=> , 
	ErrorID=> );
	
mc_Halt(
	Axis:= ax, 
	Execute:= , 
	Deceleration:= 60, 
	Jerk:= , 
	BufferMode:= , 
	Options:= , 
	Done=> , 
	Busy=> , 
	Active=> , 
	CommandAborted=> , 
	Error=> , 
	ErrorID=> );
	
Timer(IN:= , PT:= T#1S, Q=> , ET=> );


//Originalcode funktioniert wenn hier die Flanke kontrolliert wird 
//Anstelle vom Power.Status
//IF NOT mc_Power.Status THEN
//	nState:=0;
//END_IF

IF NOT bEnable THEN
	nState :=0;
END_IF

CASE nState OF 
	0:
	eState:=eBetriebszustand.Off;
	mc_power.Enable :=TRUE;
	mc_Power.Enable_Positive :=TRUE;
	
	IF bEnable AND NOT mc_power.Status THEN
		nState :=10;
	ELSIF mc_power.Status AND bEnable THEN
		nState:=20;
	END_IF
	
	10: // init Reset
	eState:=eBetriebszustand.Init;
	
	//nicht power resetten sonst durch if vor case in dauerschleife zwischen 0 und 11
	//mc_Power.Enable:=FALSE;
	//mc_Power.Enable_Positive:=FALSE;
	
	mc_Reset.Execute:=TRUE;
	
	IF mc_Reset.Done THEN
		nState:=11;
		mc_Reset.Execute:=FALSE;
	END_IF
	
	11: // init Power
	eState:=eBetriebszustand.Init;
	mc_Power.Enable:=TRUE;
	mc_Power.Enable_Positive :=TRUE;
	
	IF mc_Power.Status THEN
		nState:=20;
	END_IF
	
	20: // Ready
	eState:= eBetriebszustand.Ready;
	
	IF bExecute THEN 
		nState:=30;
	END_IF
 
	30: // Kontinuierliche Bewegung
	eState:=eBetriebszustand.Production;
	mc_Velocity.Execute:=TRUE;
	
	IF bHalt THEN 
		nState :=31;
	END_IF
	
	31: //TON verzögerung sodass Flasche noch bis zum Anschlag fährt
	eState :=eBetriebszustand.Production;
	Timer.IN:=TRUE;
	
	IF Timer.Q THEN
		nState:=32;
		Timer.IN:=FALSE;
	END_IF
	
	32: //Halten
	eState := eBetriebszustand.Production;
	mc_Velocity.Execute:=FALSE;
	mc_Halt.Execute:=TRUE;
	
	IF mc_Halt.Done THEN 
		nState:=40;
	END_IF
	
	40: // Fertig
	eState :=eBetriebszustand.Done;
	mc_halt.Execute:=FALSE;
	
	IF NOT bExecute THEN 
		nState:=20;
	END_IF
END_CASE

END_FUNCTION_BLOCK

// ---- POUs/Transport/FB_Transport_A.TcPOU
FUNCTION_BLOCK FB_Transport_A
VAR_INPUT
	bStop1 :BOOL;
	bStop2 :BOOL;
	bStop3 :BOOL;
END_VAR
VAR_OUTPUT
	//Hardware Outputs
	bStopper1 :BOOL;
	bStopper2 :BOOL;
	bStopper3 :BOOL;
END_VAR
VAR
END_VAR

bStopper1 :=  bStop1;
bStopper2 :=  bStop2;
bStopper3 :=  bStop3;

END_FUNCTION_BLOCK

// ---- POUs/Abfüllmodul/FB_EZylinder.TcPOU
FUNCTION_BLOCK FB_EZylinder
VAR_INPUT
	bGate :BOOL;
	bError :BOOL;
END_VAR
VAR_OUTPUT
	bR1 :BOOL;
	bR2 :BOOL;
END_VAR
VAR
END_VAR

bR1 :=bGate;
bR2 := NOT bGate;

IF bError THEN
	bR1 := FALSE;
	bR2 := FALSE;
END_IF

END_FUNCTION_BLOCK

// ---- POUs/FB_MqttPublisher.TcPOU
FUNCTION_BLOCK FB_MqttPublisher
VAR_INPUT
     bEnableMqtt : BOOL := TRUE;

    iBandFullmenge1 : INT;

    bEnable : BOOL;
    bExecute : BOOL;

    bEinzelSens1 : BOOL;
    bEinzelSens2 : BOOL;
    bEinzelSens3 : BOOL;

    bBandSens1 : BOOL;
    bBandSens2 : BOOL;
    bBandSens3 : BOOL;
    bBandSens4 : BOOL;

    rPcntFillLevel : REAL;
    iFillLevel1 : UINT;
    iFillLevel2 : UINT;
    iFillLevel3 : UINT;
END_VAR

VAR_OUTPUT
    bConnected : BOOL;
    bError : BOOL;
    hrErrorCode : HRESULT;
END_VAR

VAR
    fbMqttClient : FB_IotMqttClient;

    bSetParameter : BOOL := TRUE;
    bMetaSent : BOOL := FALSE;

    fbTimerPublish : TON := (PT := T#10S);

    nSendStep : INT := 0;

    sTopic : STRING(255);
    sPayload : STRING(255);

    bPublishResult : BOOL;
END_VAR

// ------------------------------------------------------------
// 1. MQTT-Verbindungsparameter einmalig setzen
// ------------------------------------------------------------
IF bSetParameter THEN
    bSetParameter := FALSE;

    fbMqttClient.sClientId := 'vier_gewinnt';
    fbMqttClient.sHostName := '158.180.44.197';
    fbMqttClient.nHostPort := 1883;
    fbMqttClient.sUserName := 'bobm';
    fbMqttClient.sUserPassword := 'letmein';
    fbMqttClient.nKeepAlive := 60;
END_IF


// ------------------------------------------------------------
// 2. MQTT-Client zyklisch ausführen
// Wichtig: Execute muss in jedem SPS-Zyklus aufgerufen werden
// ------------------------------------------------------------
fbMqttClient.Execute(bEnable);


// Status nach außen geben
bConnected := fbMqttClient.bConnected;
bError := fbMqttClient.bError;
hrErrorCode := fbMqttClient.hrErrorCode;


// ------------------------------------------------------------
// 3. Wenn Verbindung steht: Metadaten und Messwerte senden
// ------------------------------------------------------------
IF fbMqttClient.bConnected THEN

    // Metadaten einmalig nach Verbindungsaufbau senden
    IF NOT bMetaSent AND (nSendStep = 0) THEN
        nSendStep := 1;
    END_IF

    // Wenn Metadaten gesendet wurden: alle 10 Sekunden Messwerte senden
    fbTimerPublish(
        IN := bMetaSent AND (nSendStep = 0),
        PT := T#10S
    );

    IF fbTimerPublish.Q AND (nSendStep = 0) THEN
        nSendStep := 10;
    END_IF


    // --------------------------------------------------------
    // 4. Senden als kleine Schrittkette
    // Pro SPS-Zyklus wird eine MQTT-Nachricht gesendet.
    // Das ist übersichtlicher und stabiler als alles auf einmal.
    // --------------------------------------------------------
    CASE nSendStep OF

        // -------------------------
        // Einmalige retained Metadaten
        // -------------------------

        1:
            sTopic := 'aut/SoSe26/vier_gewinnt/$$groupsname';
            sPayload := 'vier_gewinnt';

            bPublishResult := fbMqttClient.Publish(
                sTopic := sTopic,
                pPayload := ADR(sPayload),
                nPayloadSize := TO_UDINT(LEN(sPayload)),
                eQoS := TcIotMqttQos.AtMostOnceDelivery,
                bRetain := TRUE,
                bQueue := TRUE
            );

            nSendStep := 2;


        2:
            sTopic := 'aut/SoSe26/vier_gewinnt/names';
            sPayload := 'Brieger, Kramer, Gneuss';

            bPublishResult := fbMqttClient.Publish(
                sTopic := sTopic,
                pPayload := ADR(sPayload),
                nPayloadSize := TO_UDINT(LEN(sPayload)),
                eQoS := TcIotMqttQos.AtMostOnceDelivery,
                bRetain := TRUE,
                bQueue := TRUE
            );

            nSendStep := 3;


        3:
            sTopic := 'aut/SoSe26/vier_gewinnt/iBandFullmenge1/$$unit';
            sPayload := '1';

            bPublishResult := fbMqttClient.Publish(
                sTopic := sTopic,
                pPayload := ADR(sPayload),
                nPayloadSize := TO_UDINT(LEN(sPayload)),
                eQoS := TcIotMqttQos.AtMostOnceDelivery,
                bRetain := TRUE,
                bQueue := TRUE
            );

            nSendStep := 4;


        4:
            sTopic := 'aut/SoSe26/vier_gewinnt/rPcntFillLevel/$$unit';
            sPayload := '%';

            bPublishResult := fbMqttClient.Publish(
                sTopic := sTopic,
                pPayload := ADR(sPayload),
                nPayloadSize := TO_UDINT(LEN(sPayload)),
                eQoS := TcIotMqttQos.AtMostOnceDelivery,
                bRetain := TRUE,
                bQueue := TRUE
            );

            nSendStep := 5;


        5:
            sTopic := 'aut/SoSe26/vier_gewinnt/iFillLevel1/$$unit';
            sPayload := '1';

            bPublishResult := fbMqttClient.Publish(
                sTopic := sTopic,
                pPayload := ADR(sPayload),
                nPayloadSize := TO_UDINT(LEN(sPayload)),
                eQoS := TcIotMqttQos.AtMostOnceDelivery,
                bRetain := TRUE,
                bQueue := TRUE
            );

            nSendStep := 6;

        6:
            sTopic := 'aut/SoSe26/vier_gewinnt/iFillLevel2/$$unit';
            sPayload := '1';

            bPublishResult := fbMqttClient.Publish(
                sTopic := sTopic,
                pPayload := ADR(sPayload),
                nPayloadSize := TO_UDINT(LEN(sPayload)),
                eQoS := TcIotMqttQos.AtMostOnceDelivery,
                bRetain := TRUE,
                bQueue := TRUE
            );

            nSendStep := 7;

        7:
            sTopic := 'aut/SoSe26/vier_gewinnt/iFillLevel3/$$unit';
            sPayload := '1';

            bPublishResult := fbMqttClient.Publish(
                sTopic := sTopic,
                pPayload := ADR(sPayload),
                nPayloadSize := TO_UDINT(LEN(sPayload)),
                eQoS := TcIotMqttQos.AtMostOnceDelivery,
                bRetain := TRUE,
                bQueue := TRUE
            );

            bMetaSent := TRUE;
            nSendStep := 0;


        // -------------------------
        // Periodische Messwerte alle 10 Sekunden
        // -------------------------

        10:
            sTopic := 'aut/SoSe26/vier_gewinnt/iFillLevel1';
            sPayload := UINT_TO_STRING(iFillLevel1);

            bPublishResult := fbMqttClient.Publish(
                sTopic := sTopic,
                pPayload := ADR(sPayload),
                nPayloadSize := TO_UDINT(LEN(sPayload)),
                eQoS := TcIotMqttQos.AtMostOnceDelivery,
                bRetain := TRUE,
                bQueue := TRUE
            );

            nSendStep := 22;


        22:
            sTopic := 'aut/SoSe26/vier_gewinnt/iFillLevel2';
            sPayload := UINT_TO_STRING(iFillLevel2);

            bPublishResult := fbMqttClient.Publish(
                sTopic := sTopic,
                pPayload := ADR(sPayload),
                nPayloadSize := TO_UDINT(LEN(sPayload)),
                eQoS := TcIotMqttQos.AtMostOnceDelivery,
                bRetain := TRUE,
                bQueue := TRUE
            );

            nSendStep := 23;


        23:
            sTopic := 'aut/SoSe26/vier_gewinnt/iFillLevel3';
            sPayload := UINT_TO_STRING(iFillLevel3);

            bPublishResult := fbMqttClient.Publish(
                sTopic := sTopic,
                pPayload := ADR(sPayload),
                nPayloadSize := TO_UDINT(LEN(sPayload)),
                eQoS := TcIotMqttQos.AtMostOnceDelivery,
                bRetain := TRUE,
                bQueue := TRUE
            );

            nSendStep := 24;


        24:
            sTopic := 'aut/SoSe26/vier_gewinnt/iBandFullmenge1';
            sPayload := INT_TO_STRING(iBandFullmenge1);

            bPublishResult := fbMqttClient.Publish(
                sTopic := sTopic,
                pPayload := ADR(sPayload),
                nPayloadSize := TO_UDINT(LEN(sPayload)),
                eQoS := TcIotMqttQos.AtMostOnceDelivery,
                bRetain := TRUE,
                bQueue := TRUE
            );

            nSendStep := 25;


        25:
            sTopic := 'aut/SoSe26/vier_gewinnt/rPcntFillLevel';
            sPayload := REAL_TO_STRING(rPcntFillLevel);

            bPublishResult := fbMqttClient.Publish(
                sTopic := sTopic,
                pPayload := ADR(sPayload),
                nPayloadSize := TO_UDINT(LEN(sPayload)),
                eQoS := TcIotMqttQos.AtMostOnceDelivery,
                bRetain := TRUE,
                bQueue := TRUE
            );

            nSendStep := 0;

    END_CASE

END_IF

END_FUNCTION_BLOCK

// ---- POUs/Extruder/FB_System_FlaschenFullstand.TcPOU
FUNCTION_BLOCK FB_System_FlaschenFullstand
VAR_INPUT
	rFilling1 : LREAL;
	rFilling2 : LREAL;
	rFilling3 : LREAL;
	Reset : BOOL;
END_VAR
VAR_OUTPUT
	rPcntFillLevelOut : REAL;
    iFillLevel1Out : UINT;
    iFillLevel2Out : UINT;
    iFillLevel3Out : UINT;
END_VAR
VAR
	rPcntFillLevel : REAL;
	rFilling1Alt : REAL;
	rFilling2Alt : REAL;
	rFilling3Alt : REAL;
	iFillLevel1 : UINT;
	iFillLevel2 : UINT;
	iFillLevel3 : UINT;
END_VAR

IF Reset THEN
	rPcntFillLevel := 0.0;
	iFillLevel1 := 0;
	iFillLevel2 := 0;
	iFillLevel3 := 0;
END_IF

IF rFilling1 <> rFilling1Alt THEN 
	rPcntFillLevel := rPcntFillLevel + (rFilling1 - rFilling1Alt)/360*7;
	iFillLevel1 := TO_UINT(rPcntFillLevel * 0.25);
ELSIF rFilling2 <> rFilling2Alt THEN
	rPcntFillLevel := rPcntFillLevel + (rFilling2 - rFilling2Alt)/360*7;
	iFillLevel2 := TO_UINT(rPcntFillLevel * 0.25)-iFillLevel1;
ELSIF rFilling3 <> rFilling3Alt THEN
	rPcntFillLevel := rPcntFillLevel + (rFilling3 - rFilling3Alt)/360*7;
	iFillLevel3 := TO_UINT(rPcntFillLevel * 0.25)- iFillLevel2-iFillLevel1;
END_IF

rFilling1Alt := rFilling1;
rFilling2Alt := rFilling2;
rFilling3Alt := rFilling3;

IF rPcntFillLevel > 100 THEN
	rPcntFillLevel := 100.0;
END_IF

rPcntFillLevelOut := rPcntFillLevel;
iFillLevel1Out := iFillLevel1;
iFillLevel2Out := iFillLevel2;
iFillLevel3Out := iFillLevel3;

END_FUNCTION_BLOCK

// ---- POUs/FUN_Scale.TcPOU
FUNCTION FUN_Scale : REAL
VAR_INPUT
	ix :UINT;
	ix_max :REAL;
	ix_min :REAL;
	ry_min :REAL;
	ry_max :REAL;
END_VAR
VAR
	rk :REAL :=0.0854492188; //für Dispenser Ultraschallsensor 
	rd :REAL :=0;
END_VAR

//FUN keine deklarierung im Hauptprogramm

rk:=(ry_max-ry_min)/(ix_max-ix_min);
rd:=ry_min-rk*ix_min;

FUN_Scale := rk*ix+rd;

IF FUN_Scale > ry_max THEN
	FUN_Scale:=ry_max;
ELSIF FUN_Scale < ry_min THEN
	FUN_Scale:=ry_min;
END_IF

END_FUNCTION

// ---- POUs/Manipulator/Roboter/FB_Roboter_Axis.TcPOU
FUNCTION_BLOCK FB_Roboter_Axis
VAR_INPUT
	bEnable :BOOL;
	bExecute :BOOL;
	rPosition :REAL;
	bRefSens :BOOL;
END_VAR
VAR_OUTPUT
	eState :eBetriebszustand;
END_VAR
VAR
	nState:INT :=0;
	mc_Reset :MC_Reset;
	mc_MoveAbsolute :MC_MoveAbsolute;
	mc_Home :MC_Home;
	mc_Power :MC_Power;
	mc_HomingMode1: MC_HomingMode;
	
END_VAR
VAR_IN_OUT
	ax :AXIS_REF;
END_VAR

ax.ReadStatus();


mc_Home(
	Axis:= ax, 
	Execute:= , 
	Position:= 0, 
	HomingMode:= mc_HomingMode1, 
	BufferMode:= , 
	Options:= , 
	bCalibrationCam:= bRefSens, 
	Done=> , 
	Busy=> , 
	Active=> , 
	CommandAborted=> , 
	Error=> , 
	ErrorID=> );
	
mc_MoveAbsolute(
	Axis:= ax, 
	Execute:= , 
	Position:= , 
	Velocity:= 30, 
	Acceleration:= 30, 
	Deceleration:= 30, 
	Jerk:= , 
	BufferMode:= , 
	Options:= , 
	Done=> , 
	Busy=> , 
	Active=> , 
	CommandAborted=> , 
	Error=> , 
	ErrorID=> );

mc_Power(
	Axis:= ax, 
	Enable:= , 
	Enable_Positive:= , 
	Enable_Negative:= , 
	Override:= , 
	BufferMode:= , 
	Options:= , 
	Status=> , 
	Busy=> , 
	Error=> , 
	ErrorID=> );
	
mc_Reset(
	Axis:= ax, 
	Execute:= , 
	Done=> , 
	Busy=> , 
	Error=> , 
	ErrorID=> );

IF NOT bEnable THEN
	nState :=0;
END_IF

CASE nState OF 
	0:
	eState:=eBetriebszustand.Off;
	mc_Power.Enable :=TRUE;
	mc_Power.Enable_Positive := TRUE;  
	mc_Power.Enable_Negative := TRUE;

	
	
	IF bEnable AND NOT mc_power.Status THEN
		nState :=10;
	ELSIF mc_power.Status AND bEnable THEN
		nState:=12;
	END_IF
	
	10: // init Reset
	eState:=eBetriebszustand.Init;
	mc_Reset.Execute:=TRUE;
	
	IF mc_Reset.Done THEN
		nState:=11;
		mc_Reset.Execute:=FALSE;
	END_IF
	
	11: // init Power
	eState:=eBetriebszustand.Init;
	
	mc_Power.Enable :=TRUE;	
	
	IF mc_Power.Status THEN
		nState:=12;
	END_IF
	
	12://Homed?
	eState:=eBetriebszustand.Init;
	
	IF ax.Status.Homed THEN
		nstate:=20;
	ELSE
		nstate:=13;
	END_IF
	
	13://Homing
	eState:=eBetriebszustand.Init;
	
	mc_Home.Execute :=TRUE;
	
	IF mc_Home.Done THEN
		mc_Home.Execute :=FALSE;
		nstate:= 20;
	END_IF
	
	
	20: // Ready
	eState:= eBetriebszustand.Ready;
	
	IF bExecute THEN 
		nState:=30;
	END_IF
 
	30: // Bewegung
	eState:=eBetriebszustand.Production;
	mc_MoveAbsolute.Position := rPosition;
	mc_MoveAbsolute.Execute :=TRUE;
	
	IF mc_MoveAbsolute.Done THEN 
		mc_MoveAbsolute.Execute:=FALSE;
		nState :=40;
	END_IF
	
	40: // Fertig
	eState :=eBetriebszustand.Done;
	
	IF NOT bExecute THEN 
		nState:=20;
	END_IF

END_CASE

END_FUNCTION_BLOCK

// ---- POUs/Manipulator/Roboter/FB_Roboter_E.TcPOU
FUNCTION_BLOCK FB_Roboter_E
VAR_INPUT
	bRefMax_in :BOOL;
	bRefMin_in :BOOL;
	
END_VAR
VAR_OUTPUT
	bRefMax_out :BOOL;
	bRefMin_out :BOOL;
	
END_VAR
VAR
END_VAR

bRefMax_out :=  NOT bRefMax_in;
bRefMin_out := NOT bRefMin_in;

END_FUNCTION_BLOCK

// ---- POUs/Manipulator/Roboter/FB_Roboter_Logik.TcPOU
FUNCTION_BLOCK FB_Roboter_Logik
VAR_INPUT
	bEnable :BOOL;
	bExecute :BOOL;

	pPositionX :REAL;
	bRefmin_X :BOOL;
	bRefmax_X :BOOL;
	
	pPositionY :REAL;
	bRefmin_Y :BOOL;
	bRefmax_Y :BOOL;
	
	pPositionZ :REAL;
	bRefmin_Z :BOOL;
	bRefmax_Z :BOOL;
	
	
	
	
END_VAR
VAR_OUTPUT
	bBreak :BOOL;
	
	
	eState :eBetriebszustand;
	
END_VAR
VAR
	fb_Roboter_Axis_X : FB_Roboter_Axis;
	fb_Roboter_Axis_Y : FB_Roboter_Axis;
	fb_Roboter_Axis_Z : FB_Roboter_Axis;
	//fb_Roboter_Gripper : FB_Roboter_Axis;
	
	nState :INT;
END_VAR

//soft limits bei Achse selbst für realen Betrieb einstellen 

fb_Roboter_Axis_X(
	bEnable:= , 
	bExecute:= , 
	rPosition:= , 
	bRefSens:= bRefmin_X, 
	eState=> , 
	ax:= IFC_HW.ax_ManX);
fb_Roboter_Axis_Y(
	bEnable:= , 
	bExecute:= , 
	rPosition:= , 
	bRefSens:= bRefmin_Y, 
	eState=> , 
	ax:= IFC_HW.ax_ManY);
fb_Roboter_Axis_Z(
	bEnable:= , 
	bExecute:= , 
	rPosition:= , 
	bRefSens:= bRefmin_Z, 
	eState=> , 
	ax:= IFC_HW.ax_ManZ);

IF NOT bEnable THEN
	nState :=0;
END_IF

CASE nState OF
	0: //off
	eState := eBetriebszustand.Off;
	
	IF bEnable THEN
		nstate :=1;
	END_IF
	
	1: //init
	eState := eBetriebszustand.Init;
	fb_Roboter_Axis_X.bEnable := TRUE;
	fb_Roboter_Axis_Y.bEnable := TRUE;
	fb_Roboter_Axis_Z.bEnable := TRUE;
	
	IF (fb_Roboter_Axis_X.eState = eBetriebszustand.Ready) AND (fb_Roboter_Axis_Y.eState = eBetriebszustand.Ready) AND (fb_Roboter_Axis_Z.eState = eBetriebszustand.Ready) THEN 
		nstate :=2;
	END_IF
	
	2: //Ready
	eState := eBetriebszustand.Ready;
	
	IF bExecute THEN 
		nstate :=21;
	END_IF
	
	21: //check z hight
	eState := eBetriebszustand.Production;
	
	IF IFC_HW.ax_ManZ.NcToPlc.ActPos > GVL_PosKinematic.pZoff THEN
		nstate :=22;
	ELSE
		nstate :=23;
	END_IF
	
	22: //Move Z to safe position
	eState := eBetriebszustand.Production;
	
	fb_Roboter_Axis_Z.rPosition :=45;
	fb_Roboter_Axis_Z.bExecute :=TRUE;
	bBreak :=TRUE;
	
	IF fb_Roboter_Axis_Z.eState = eBetriebszustand.Done THEN
		fb_Roboter_Axis_Z.bExecute :=FALSE;
		bBreak :=FALSE;
		nstate :=23;
	END_IF
	
	23: //Move xy
	eState := eBetriebszustand.Production;
	
	fb_Roboter_Axis_X.rPosition :=pPositionX;
	fb_Roboter_Axis_X.bExecute :=TRUE;
	fb_Roboter_Axis_Y.rPosition :=pPositionY;
	fb_Roboter_Axis_Y.bExecute :=TRUE;
	
	IF (fb_Roboter_Axis_X.eState = eBetriebszustand.Done) AND (fb_Roboter_Axis_Y.eState = eBetriebszustand.Done) THEN
		fb_Roboter_Axis_X.bExecute :=FALSE;
		fb_Roboter_Axis_Y.bExecute :=FALSE;
		nstate :=24;
	END_IF
	
	24: //Move Z
	eState := eBetriebszustand.Production;
	
	fb_Roboter_Axis_Z.rPosition :=pPositionZ;
	fb_Roboter_Axis_Z.bExecute :=TRUE;
	bBreak :=TRUE;
	
	IF fb_Roboter_Axis_Z.eState = eBetriebszustand.Done THEN
		fb_Roboter_Axis_Z.bExecute :=FALSE;
		bBreak :=FALSE;
		nstate :=25;
	END_IF
	
	25: //Done
	eState := eBetriebszustand.Done;
	
	IF NOT bExecute THEN
		nstate :=2;
	END_IF
	
	
END_CASE

END_FUNCTION_BLOCK

// ---- VISUs/Visualization.TcVIS
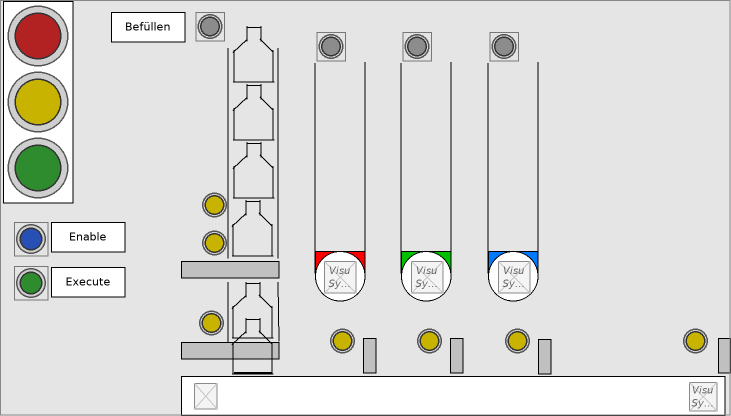
VISUALIZATION Visualization  // 731x416
    Rectangle (315,251 50x24)
        p2773130477: - MAIN.fbExt1.iFillLevel
    Lamp1 (200,190 29x30), variable: MAIN.bOut_VereinzelungNS1, style: Lamp-Lamp1-Yellow
    Lamp1 (200,228 29x30), variable: MAIN.bOut_VereinzelungNS2, style: Lamp-Lamp1-Yellow
    Lamp1 (197,308 29x30), variable: MAIN.bOut_VereinzelungNS3, style: Lamp-Lamp1-Yellow
    Group (3,1 70x202)
        Rectangle (0,0 70x202)
        Lamp1 (0,0 70x70), variable: bAmpelRot, style: Lamp-Lamp1-Red
        Lamp1 (0,66 70x70), variable: bAmpelGelb, style: Lamp-Lamp1-Yellow
        Lamp1 (0,132 70x70), variable: bAmpelGrun, style: Lamp-Lamp1-Green
    Line (228,258) (228,48)
    Line (278,258) (278,48)
    Line (279,341) (278,282)
    Line (228,342) (228,282)
    Rectangle (181,261 98x17)
        p3528305787: MAIN.fbVereinzelung.S1pos
        p874137650: MAIN.fbVereinzelung.S1pos
    Rectangle (181,342 98x17)
        p3528305787: MAIN.fbVereinzelung.S2pos
        p874137650: MAIN.fbVereinzelung.S2pos
    PushSwitch (12,222 38x34), variable: bEnable, behaviour: TOGGLE, style: Switch-PushSwitch-Blue
    PushSwitch (12,266 38x34), variable: bExecute, behaviour: TAP, style: Switch-PushSwitch-Green
    Rectangle (51,222 74x30), "Enable"
    Rectangle (51,267 74x30), "Execute"
    Group (232,200 41x57), invisible if: not MAIN.fbVereinzelung.fbSpeicherRohr.aSpeicher[0]
        Line (1,56) (1,24)
        Line (40,55) (40,24)
        Line (41,56) (0,56)
        Line (0,26) (14,13)
        Line (40,26) (27,13)
        Line (14,15) (14,0)
        Line (28,15) (28,0)
        Line (14,1) (28,1)
    Group (233,142 41x57), invisible if: Not MAIN.fbVereinzelung.fbSpeicherRohr.aSpeicher[1]
        Line (1,56) (1,24)
        Line (40,55) (40,24)
        Line (41,56) (0,56)
        Line (0,26) (14,13)
        Line (40,26) (27,13)
        Line (14,15) (14,0)
        Line (28,15) (28,0)
        Line (14,1) (28,1)
    Group (232,282 41x57), invisible if: not MAIN.bOut_VereinzelungNS3
        Line (1,56) (1,24)
        Line (40,55) (40,24)
        Line (41,56) (0,56)
        Line (0,26) (14,13)
        Line (40,26) (27,13)
        Line (14,15) (14,0)
        Line (28,15) (28,0)
        Line (14,1) (28,1)
    Group (233,84 41x57), invisible if: Not MAIN.fbVereinzelung.fbSpeicherRohr.aSpeicher[2]
        Line (1,56) (1,24)
        Line (40,55) (40,24)
        Line (41,56) (0,56)
        Line (0,26) (14,13)
        Line (40,26) (27,13)
        Line (14,15) (14,0)
        Line (28,15) (28,0)
        Line (14,1) (28,1)
    Group (233,26 41x57), invisible if: Not MAIN.fbVereinzelung.fbSpeicherRohr.aSpeicher[3]
        Line (1,56) (1,24)
        Line (40,55) (40,24)
        Line (41,56) (0,56)
        Line (0,26) (14,13)
        Line (40,26) (27,13)
        Line (14,15) (14,0)
        Line (28,15) (28,0)
        Line (14,1) (28,1)
    PushSwitch (194,12 32x29), variable: MAIN.fbVereinzelung.bBefullen, behaviour: TAP, style: Switch-PushSwitch-Gray
    RoundedRectangle (181,376 544x40)
    Lamp1 (328,326 29x30), variable: MAIN.bOUT_CnvNS1, style: Lamp-Lamp1-Yellow
    Lamp1 (503,326 29x30), variable: MAIN.bOUT_CnvNS3, style: Lamp-Lamp1-Yellow
    Lamp1 (415,326 29x30), variable: MAIN.bOUT_CnvNS2, style: Lamp-Lamp1-Yellow
    Lamp1 (681,326 29x30), variable: MAIN.bOUT_CnvNS4, style: Lamp-Lamp1-Yellow
    Group (232,318 41x57), invisible if: not MAIN.fbCNV.bBottleOnCNV
        p3560616238: MAIN.fbCNV.iBottlePos
        Line (1,56) (1,24)
        Line (40,55) (40,24)
        Line (41,56) (0,56)
        Line (0,26) (14,13)
        Line (40,26) (27,13)
        Line (14,15) (14,0)
        Line (28,15) (28,0)
        Line (14,1) (28,1)
    Rectangle (363,338 13x35), invisible if: MAIN.bIN_Stopper1
    Rectangle (450,338 13x35), invisible if: MAIN.bIN_Stopper2
    Rectangle (538,339 13x35), invisible if: MAIN.bIN_Stopper3
    Rectangle (718,338 13x35)
    Image (194,383 23x26), invisible if: not MAIN.fbCNV.bCNVisMoving, image: VisuSymbols.Symbols.ArrowHalfRightUp
    Image (689,382 28x29), invisible if: not MAIN.fbCNV.bCNVisMoving, image: VisuSymbols.Symbols.ArrowHalfRightDown
    Rectangle (111,12 74x30), "Befüllen"
    Ellipse (315,251 50x50)
    Line (315,273) (315,63)
    Line (365,272) (365,62)
    Rectangle (401,251 50x24)
        p2773130477: - MAIN.fbExt2.iFillLevel
    Ellipse (401,251 50x50)
    Line (401,273) (401,63)
    Line (451,272) (451,62)
    Rectangle (488,251 50x24)
        p2773130477: - MAIN.fbExt3.iFillLevel
    Ellipse (488,251 50x50)
    Line (488,273) (488,63)
    Line (538,272) (538,62)
    PushSwitch (315,32 32x29), variable: MAIN.bRefill1, behaviour: TAP, style: Switch-PushSwitch-Gray
    PushSwitch (401,32 32x29), variable: MAIN.bRefill2, behaviour: TAP, style: Switch-PushSwitch-Gray
    PushSwitch (488,32 32x29), variable: MAIN.bRefill3, behaviour: TAP, style: Switch-PushSwitch-Gray
    Image (324,261 32x32), invisible if: MAIN.fbExt1.NotMoving, image: VisuSymbols.Symbols.ArrowCircle2RightRightLeft
    Image (411,261 32x32), invisible if: MAIN.fbExt2.NotMoving, image: VisuSymbols.Symbols.ArrowCircle2RightRightLeft
    Image (498,261 32x32), invisible if: MAIN.fbExt3.NotMoving, image: VisuSymbols.Symbols.ArrowCircle2RightRightLeft
    Rectangle (234,372 38x1), invisible if: not MAIN.fbCNV.bBottleOnCNV
        p2773130477: - MAIN.fbBottleLevel.iFillLevel3 - MAIN.fbBottleLevel.iFillLevel1 - MAIN.fbBottleLevel.iFillLevel2
        p3560616238: MAIN.fbCNV.iBottlePos
        p1126004900: - MAIN.fbBottleLevel.iFillLevel1 - MAIN.fbBottleLevel.iFillLevel2
    Rectangle (234,372 38x1), invisible if: not MAIN.fbCNV.bBottleOnCNV
        p2773130477: - MAIN.fbBottleLevel.iFillLevel2 - MAIN.fbBottleLevel.iFillLevel1
        p3560616238: MAIN.fbCNV.iBottlePos
        p1126004900: - MAIN.fbBottleLevel.iFillLevel1
    Rectangle (234,372 38x1), invisible if: not MAIN.fbCNV.bBottleOnCNV
        p2773130477: - MAIN.fbBottleLevel.iFillLevel1
        p3560616238: MAIN.fbCNV.iBottlePos
END_VISUALIZATION
